Staubli VAL3: ENTRYBOX.dtx

num nDummy
num nFocused
num nLblPosX[3]
  [1] = 22
num nLblPosY[3] = 6
public num nNumOfLabel = 3
public num nNumOfTxtBox = 10
num nPageUpCol
num nPageUpRow
num nTxtFocused
num nTxtMaxVal[10]
  [0] = 1000
  [1] = 1000
  [2] = 200
  [4] = 200
  [5] = 20
  [6] = 99
  [8] = 999
  [9] = 999
num nTxtMinVal[10]
  [0] = -1000
  [1] = -1000
  [2] = 5
  [4] = 1
  [5] = 1
  [6] = 1
num nTxtPosX[10]
  [6] = 22
  [7] = 22
  [8] = 22
  [9] = 22
num nTxtPosY[10]
  [0] = 1
  [1] = 2
  [2] = 3
  [3] = 4
  [4] = 7
  [5] = 8
  [6] = 1
  [7] = 3
  [8] = 4
  [9] = 5
num nVIDEOCUSTOM = 2
num nVIDEOINVERSED = 1
num nVIDEONORMAL
string sErrMsgList[6]
  [1] = "The library *\../* couldn't not be loaded because of the error code n°*"
  [2] = "Error from definition library *\../*."
  [3] = "The variable sListItem* of the definition library is not defined."
  [4] = "The  caption '*\../*'  does not exist"
string sErrorMessage = "The library GenericWin couldn't not be loaded because of the error code n°30"
string sListItems
bool bDrawFrame
public mdesc mNomSpeed = {blend=off}
